FUNCTION_BLOCK "Alarm"
{ S7_Optimized_Access := 'TRUE' }
AUTHOR : Searinox
VERSION : 0.1
   VAR_INPUT
      iCvOff : Bool;   // Control Voltage Off / emergency stop
      iFuseOutputsErr : Bool;   // Fuse Outputs Error
      iCt1RepairSwitchOff : Bool;   // Cooling Tower 1 Repair Switch
      iCt2RepairSwitchOff : Bool;   // Cooling Tower 2 Repair Switch
      iFan1 : "Fan";
      iFan2 : "Fan";
      iPumpPlant1 : "Pump";
      iPumpPlant2 : "Pump";
      iPumpCoolWater1 : "Pump";
      iPumpCoolWater2 : "Pump";
      iPumpFurnace1 : "Pump";
      iPumpFurnace2 : "Pump";
      iSprayPipe1 : "Valve";
      iSprayPipe2 : "Valve";
      iLiftingSys1 : "LiftingSys";
      iLiftingSys2 : "LiftingSys";
      iTempPlant : "Temperature";
      iTempFurnace : "Temperature";
      iSurgeTank : "Tank";
      iBleedingUnit : "BleedingUnit";
   END_VAR

   VAR_OUTPUT
      oAlarmCount : Int := 0;
      oAlarmCountCrit : Int;
      oAlarmLamp : Bool := false;
   END_VAR

   VAR
      sCvOff : Int;
      sFuseOutputsErr : Int;
      sCt1FanErr : Int;
      sCt1RepairSwitchOff : Int;
      sCt2FanErr : Int;
      sCt2RepairSwitchOff : Int;
      sFanErrCrit : Int;
      sPumpPlant1Err : Int;
      sPumpPlant2Err : Int;
      sPumpPlantErrCrit : Int;
      sPumpCoolWater1Err : Int;
      sPumpCoolWater2Err : Int;
      sPumpCoolWaterErrCrit : Int;
      sPumpFurnace1Err : Int;
      sPumpFurnace2Err : Int;
      sPumpFurnaceErrCrit : Int;
      sFlowTempPlantHot : Int;
      sFlowTempFurnaceHot : Int;
      sPressureDeltaPerc1 : Int;
      sPressureDeltaPerc2 : Int;
      sSurgeTankRunDry : Int;
      sSurgeTankOverflow : Int;
      Ton0 {OriginalPartName := 'IEC_TIMER'; LibVersion := '1.0'} : TON_TIME;
      Ton1 {OriginalPartName := 'IEC_TIMER'; LibVersion := '1.0'} : TON_TIME;
      sSprayPipeOpenTimeout1 : Int;
      sSprayPipeOpenTimeout2 : Int;
      sBleedingUnitErr : Int;
   END_VAR


BEGIN
	REGION bool
	    #sCvOff := BOOL_TO_INT(#iCvOff);
	    #sFuseOutputsErr := BOOL_TO_INT(#iFuseOutputsErr);
	    #sCt1FanErr := BOOL_TO_INT(#iFan1.HasError);
	    #sCt2FanErr := BOOL_TO_INT(#iFan2.HasError);
	    #sCt1RepairSwitchOff := BOOL_TO_INT(#iCt1RepairSwitchOff);
	    #sCt2RepairSwitchOff := BOOL_TO_INT(#iCt2RepairSwitchOff);
	    #sFanErrCrit := BOOL_TO_INT((#iFan1.HasError AND #iFan2.HasError) OR
	                                (#iCt1RepairSwitchOff AND #iCt2RepairSwitchOff));
	    #sPumpPlant1Err := BOOL_TO_INT(#iPumpPlant1.HasError);
	    #sPumpPlant2Err := BOOL_TO_INT(#iPumpPlant2.HasError);
	    #sPumpPlantErrCrit := BOOL_TO_INT(#iPumpPlant1.HasError AND #iPumpPlant2.HasError);
	    #sPumpCoolWater1Err := BOOL_TO_INT(#iPumpCoolWater1.HasError);
	    #sPumpCoolWater2Err := BOOL_TO_INT(#iPumpCoolWater2.HasError);
	    #sPumpCoolWaterErrCrit := BOOL_TO_INT(#iPumpCoolWater1.HasError AND #iPumpCoolWater2.HasError);
	    #sPumpFurnace1Err := BOOL_TO_INT(#iPumpFurnace1.HasError);
	    #sPumpFurnace2Err := BOOL_TO_INT(#iPumpFurnace2.HasError);
	    #sPumpFurnaceErrCrit := BOOL_TO_INT(#iPumpFurnace1.HasError AND #iPumpFurnace2.HasError);
	    #sBleedingUnitErr := BOOL_TO_INT(#iBleedingUnit.HasError);
	END_REGION
	REGION analog
	    // temperatures
	    #sFlowTempPlantHot := BOOL_TO_INT(#iTempPlant.Val.R >= (
	                                      #iTempPlant.SetPoint.Upper.R +
	                                      #iTempPlant.Limits.Max.R));

	    #sFlowTempFurnaceHot := BOOL_TO_INT(#iTempFurnace.Val.R >= (
	                                        #iTempFurnace.SetPoint.Upper.R +
	                                        #iTempFurnace.Limits.Max.R));
	    // pressures
	    #sPressureDeltaPerc1 := BOOL_TO_INT(#iLiftingSys1.DeltaPressure.Val.R >=
	                                        #iLiftingSys1.DeltaPressure.Limits.Max.R);

	    #sPressureDeltaPerc2 := BOOL_TO_INT(#iLiftingSys2.DeltaPressure.Val.R >=
	                                        #iLiftingSys2.DeltaPressure.Limits.Max.R);
	    // levels
	    #sSurgeTankRunDry := BOOL_TO_INT(#iSurgeTank.Val.I <=
	                                     #iSurgeTank.Limits.Min.I);

	    #sSurgeTankOverflow := BOOL_TO_INT(#iSurgeTank.Val.I >=
	                                       #iSurgeTank.Limits.Max.I);
	END_REGION
	REGION timeout
	    #Ton0(IN := #iSprayPipe1.Q,
	          PT := #iSprayPipe1.Timeout);
	    #sSprayPipeOpenTimeout1 := BOOL_TO_INT(#Ton0.Q AND NOT #iSprayPipe1.IsOpen);
	    #Ton1(IN := #iSprayPipe2.Q,
	          PT := #iSprayPipe2.Timeout);
	    #sSprayPipeOpenTimeout2 := BOOL_TO_INT(#Ton1.Q AND NOT #iSprayPipe2.IsOpen);
	END_REGION

	#oAlarmCount := 0;
	#oAlarmCount += #sCvOff;
	#oAlarmCount += #sFuseOutputsErr;
	#oAlarmCount += #sCt1FanErr;
	#oAlarmCount += #sCt1RepairSwitchOff;
	#oAlarmCount += #sCt2FanErr;
	#oAlarmCount += #sCt2RepairSwitchOff;
	#oAlarmCount += #sPumpPlant1Err;
	#oAlarmCount += #sPumpPlant2Err;
	#oAlarmCount += #sPumpCoolWater1Err;
	#oAlarmCount += #sPumpCoolWater2Err;
	#oAlarmCount += #sPumpFurnace1Err;
	#oAlarmCount += #sPumpFurnace2Err;
	#oAlarmCount += #sBleedingUnitErr;
	#oAlarmCount += #sFlowTempPlantHot;
	#oAlarmCount += #sFlowTempFurnaceHot;
	#oAlarmCount += #sPressureDeltaPerc1;
	#oAlarmCount += #sPressureDeltaPerc2;
	#oAlarmCount += #sSurgeTankRunDry;
	#oAlarmCount += #sSurgeTankOverflow;
	#oAlarmCount += #sSprayPipeOpenTimeout1;
	#oAlarmCount += #sSprayPipeOpenTimeout2;

	#oAlarmCountCrit := 0;
	#oAlarmCountCrit += #sCvOff;
	#oAlarmCountCrit += #sFuseOutputsErr;
	#oAlarmCountCrit += #sFanErrCrit;
	#oAlarmCountCrit += #sPumpPlantErrCrit;
	#oAlarmCountCrit += #sPumpCoolWaterErrCrit;
	#oAlarmCountCrit += #sPumpFurnaceErrCrit;
	#oAlarmCountCrit += #sSurgeTankRunDry;
	#oAlarmCountCrit += #sSurgeTankOverflow;

	#oAlarmLamp := #oAlarmCount > 0;

END_FUNCTION_BLOCK

